{attribute addProperty BoxType "EP1859-0042-0019"}
{attribute addProperty Id "DI_X01AT %I*ARRAY[0..1] OF DI_X_E4AEF59E429496728842949672950DI_X02AT %I*ARRAY[0..1] OF DI_X_E4AEF59E429496728842949672950DI_X03AT %I*ARRAY[0..1] OF DI_X_E4AEF59E429496728842949672950DI_X04AT %I*ARRAY[0..1] OF DI_X_E4AEF59E429496728842949672950DO_X05AT %Q*ARRAY[0..1] OF DO_X_7F374EB0429496728842949672950DO_X06AT %Q*ARRAY[0..1] OF DO_X_7F374EB0429496728842949672950DO_X07AT %Q*ARRAY[0..1] OF DO_X_7F374EB0429496728842949672950DO_X08AT %Q*ARRAY[0..1] OF DO_X_7F374EB0429496728842949672950WcStateAT %I*WcState_98A4DF7520.250InfoDataAT %I*InfoData_192954DE1620"}
{attribute addProperty CRC "3412465426"}
{attribute addProperty SizeInBites "4294967250"}
{attribute addProperty SizeInBytes "34359738362.25"}
TYPE EP1859_B48C22F8 :
STRUCT
	{attribute addProperty Name "DI_X01"}
	DI_X01 : ARRAY[0..1] OF DI_X_E4AEF59E;
	{attribute addProperty Name "DI_X02"}
	DI_X02 : ARRAY[0..1] OF DI_X_E4AEF59E;
	{attribute addProperty Name "DI_X03"}
	DI_X03 : ARRAY[0..1] OF DI_X_E4AEF59E;
	{attribute addProperty Name "DI_X04"}
	DI_X04 : ARRAY[0..1] OF DI_X_E4AEF59E;
	{attribute addProperty Name "DO_X05"}
	DO_X05 : ARRAY[0..1] OF DO_X_7F374EB0;
	{attribute addProperty Name "DO_X06"}
	DO_X06 : ARRAY[0..1] OF DO_X_7F374EB0;
	{attribute addProperty Name "DO_X07"}
	DO_X07 : ARRAY[0..1] OF DO_X_7F374EB0;
	{attribute addProperty Name "DO_X08"}
	DO_X08 : ARRAY[0..1] OF DO_X_7F374EB0;
	{attribute addProperty Name "WcState"}
	WcState : WcState_98A4DF75;
	{attribute addProperty Name "InfoData"}
	InfoData : InfoData_192954DE;
END_STRUCT
END_TYPE

(* stored: Version 1.2.0.0, ProductVersion 3.1.4024.9
   DUT EP1859_B48C22F8: Id {b333320b-cfc8-4e42-95e1-fcbfa4b1741e} *)
